FUNCTION_BLOCK ST001_ComponentsHandler EXTENDS TcoCore.TcoObject
VAR
	{attribute addProperty Name "<#PART PRESENCE SENSOR#>"}
	_partPresent : TcoElements.TcoDi(THIS^);
	{attribute addProperty Name "<#START BUTTON#>"}
    _startButton : TcoElements.TcoDi(THIS^);
	{attribute addProperty Name "<#PRESS PISTON#>"}
    _press : TcoPneumatics.TcoCylinder(THIS^);
	{attribute addProperty Name "<#ALARM OUTPUT#>"}
	_alarmOutput : TcoElements.TcoDo(THIS^);
	{attribute addProperty Name "<#DRIVE#>"}
	_drive : TcoDrivesBeckhoff.TcoDriveSimple(THIS^);
END_VAR

_partPresent(inoSignal := IO.EC001.A1.IO._1);
_startButton(inoSignal := IO.EC001.A1.IO._2);
_press(inoAtHomePos:= IO.EC001.A1.IO._3, inoAtWorkPos:= IO.EC001.A1.IO._4, inoToHomePos:= IO.EC001.A10.IO._1, inoToWorkPos:=IO.EC001.A10.IO._2);

PROPERTY PartPresent : REFERENCE TO TcoElements.TcoDi
GET
PartPresent REF= _partPresent;
END_GET
END_PROPERTY

PROPERTY Press : REFERENCE TO TcoPneumatics.TcoCylinder
GET
Press REF= _press;
END_GET
END_PROPERTY

METHOD Service
THIS^._partPresent.Service();
THIS^._startButton.Service();
THIS^._press.Service();
THIS^._alarmOutput.Service();
END_METHOD

END_FUNCTION_BLOCK

(* stored: Version 1.1.0.1, ProductVersion 3.1.4024.9
   POU ST001_ComponentsHandler: Id {e26fa0d3-d3d7-028e-3078-514e2e8d1a78}, SpecialFunc None
   Property PartPresent: Id {f5cdf153-1188-001b-0f38-1f9504216ef9}
   Get Get: Id {46de24c4-0ea6-09cd-2268-c904722ac596}
   Property Press: Id {ed012438-e4fb-0ad6-2f3f-43e788f64a37}
   Get Get: Id {75a426ad-70f8-045d-2bc3-929207cc534a}
   Method Service: Id {d9a55f5d-e4b4-0800-35fa-c2749c040034} *)
